Fanuc KAREL source: kt00373.KL

-- PROVISIONAL review KL for V1013-1; original PC SHA256 e506fae7f821949ab2b5dcc7c808490de7ecca9ce4ab55c15db7857d5d8b8faa
-- Incomplete behavior may be omitted. Consult companion uncertainty JSON. Do not deploy.
PROGRAM KT00373
%NOLOCKGROUP
VAR
  B1 : BOOLEAN
  B2 : BOOLEAN
  OUT : BOOLEAN
BEGIN
  -- UNRESOLVED_PC offsets 5-12; opcodes 9D,23
  -- UNRESOLVED_PC offsets 17-24; opcodes 9C,23
  -- UNRESOLVED_PC offsets 29-36; opcodes 9D,23
  -- UNRESOLVED_PC offsets 41-48; opcodes 9C,23
  -- UNRESOLVED_PC offsets 53-72; opcodes 21,21,5A,23
  -- UNRESOLVED_PC offsets 77-81; opcodes 7F
END KT00373
